FUNCTION_BLOCK bfb_off_peak_types
  (* Standard: 61499-2 *)
  (* Version 0.1, 2018-00-11, palme, DESKTOP-TGOEKBD *)
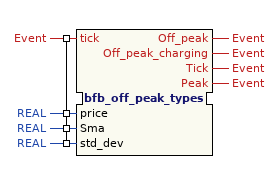
  EVENT_INPUT
    tick WITH price, Sma, std_dev;
  END_EVENT
  EVENT_OUTPUT
    Off_peak;
    Off_peak_charging;
    Tick;
    Peak;
  END_EVENT
  VAR_INPUT
    price : REAL;
    Sma : REAL;
    std_dev : REAL;
  END_VAR
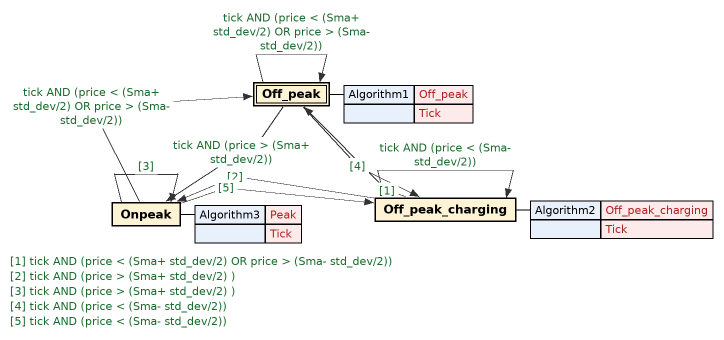
  EC_STATES
    Off_peak : Algorithm1 -> Off_peak, -> Tick;
    Off_peak_charging : Algorithm2 -> Off_peak_charging, -> Tick;
    Onpeak : Algorithm3 -> Peak, -> Tick;
  END_STATES
  EC_TRANSITIONS
    Off_peak TO Off_peak_charging := tick AND (price < (Sma- std_dev/2));
    Off_peak TO Off_peak := tick AND (price < (Sma+ std_dev/2) OR price > (Sma- std_dev/2));
    Off_peak TO Onpeak := tick AND (price > (Sma+ std_dev/2));
    Off_peak_charging TO Off_peak_charging := tick AND (price < (Sma- std_dev/2));
    Off_peak_charging TO Off_peak := tick AND (price < (Sma+ std_dev/2) OR price > (Sma- std_dev/2));
    Off_peak_charging TO Onpeak := tick AND (price > (Sma+ std_dev/2) );
    Onpeak TO Off_peak := tick AND (price < (Sma+ std_dev/2) OR price > (Sma- std_dev/2));
    Onpeak TO Off_peak_charging := tick AND (price < (Sma- std_dev/2));
    Onpeak TO Onpeak := tick AND (price > (Sma+ std_dev/2) );
  END_TRANSITIONS
  ALGORITHM Algorithm1 IN C:
printf("OFF_peak in Off peak types\r\n");
  END_ALGORITHM
  ALGORITHM Algorithm2 IN C:
printf("OFF_peak CHARGING in Off peak types\r\n");
  END_ALGORITHM
  ALGORITHM Algorithm3 IN C:
printf("ON PEAK IN OFF peak types\r\n");
  END_ALGORITHM
END_FUNCTION_BLOCK
